RoboDK station: FanucCell.rdk

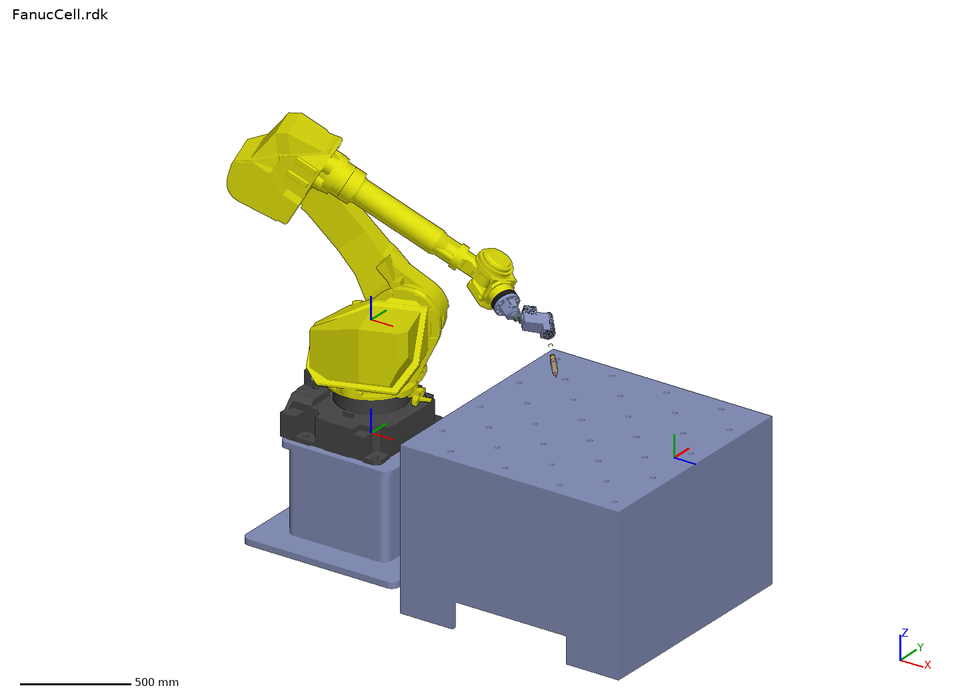
[picture v0: the station drawn from its stored meshes, robots at their saved joint values, targets as dots, program paths as lines]
Station FanucCell (saved by RoboDK 5.4.2). Poses are relative to the parent item; angles as X-Y-Z fixed-axis rotations.
  - frame RobotCell at (0, 0, 0) mm
    - object RobotStand at (42.5, -2.5, 0) mm, size 840 x 840 x 500 mm, geometry from RobotStand.STEP
    - object WeldingTable at (-75, 0, 0) mm, size 1200 x 1200 x 840 mm, geometry from WeldingTable.STEP
    - frame Fanuc M-710iC/70 Base at (0, 0, 565) mm
      - robot Fanuc M-710iC/70: 6 axes, payload 70 kg, reach 1360 mm, repeatability 0.07 mm, weight 545 kg
          modified DH rows (alpha deg, a mm, theta deg, d mm): 0, 0, 0, 570; -90, 150, -90, 0; 0, 870, 0, 0; -90, 170, 0, 1016; 90, 0, 0, 0; -90, 0, 0, 175
          base shift (0, 0, -570) mm
          joint limits [-180, -110, -65, -360, -125, -360] to [180, 110, 245, 360, 125, 360]; home [0, 0, 0, 0, 0, 0]; saved at [19.147, -41.242, -29.998, 90.079, -39.541, -16.05]
        - tool Torch, TCP at (4.87, 0, 467.95) mm, rotated rx 0 ry -22 rz 0 deg, size 234.3 x 124.1 x 483.7 mm
    - frame ItemFrame at (1660, 0, 340) mm, rotated rx 90 ry 0 rz 90 deg
